KUKA KRL program: chk_w7_wechs_ok.src

&ACCESS RV2
&COMMENT Gripper Accelo Traseiro
DEF chk_w7_wechs_ok( )

; VERIFICAÇÃO DE FERRAMENTA: GRIPPER TRASEIRO ACCELO

$TIMER[10] = 0
$TIMER_STOP[10] = FALSE

wait for (($IN[585]) and ($IN[577]) and (not $in[161]) and ($in[177]) and ($in[193]) and ( $in[169]) and ($IN[185]) and ($in[201]) and ($in[209]) AND ($in[219]))

$TIMER_STOP[10] = TRUE
$TIMER[10] = 0

;//---- End -------
;Diag_Appl(#Off,5)

END
